ABB RobotStudio station: Assignment2_task#1.rsstn

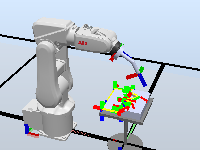
Station Assignment2_task#1 (saved by RobotStudio 20.1.9014.1)
Controller SystemTask1, task T_ROB1: task frame (RAPID world) sits at (150, 100, 0) mm in the station
Controller SystemTask1
  mechanical unit ROB_1: IRB120_3_58__01, 6 joints, base frame (0, 0, 0) mm
Layout (positions relative to the parent item):
  - IRB120_3_58__01 [mechanism, from Robots\IRB120_3_58_G_01.rslib] at (150, 100, 0) mm; joint values [0, 0, 0, 0, 0.5236, 0] (rad or m)
  - AssemblyWeldingTorch [part] at (452.8, 131.78, 541.25) mm, rotated rx -30 ry 0 rz -90 deg
  - Task1_Part1_2 [part] at (570, 0, 300) mm, rotated rx 90 ry 0 rz 0 deg
  - Task1_Part2 [part] at (470, 0, 300) mm, rotated rx 90 ry 0 rz 0 deg
  - Part_1 [part]
  - Part_2 [part]
  - Part_3 [part]
  - Part_4 [part]
Attachment: AssemblyWeldingTorch is attached to IRB120_3_58__01 / Link6
Attachment: Task1_Part2 is attached to Task1_Part1_2
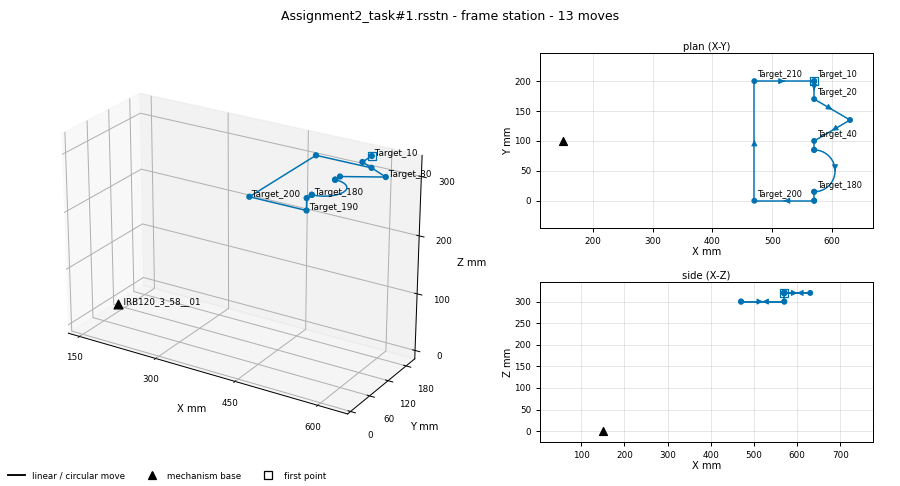
[picture p0: tool path of Assignment2_task#1.rsstn in frame station, 13 of 13 moves have a stored position in this frame; points joined in program order, loops and branches not executed]
Targets, tools, work objects and paths stored in the station, written as RAPID:
! task T_ROB1
MODULE CalibData
  TASK PERS tooldata WeldingTorch:=[TRUE,[[41,0,150.621],[0.965925826,0,0.258819045,0]],[1,[0,0,1],[1,0,0,0],0,0,0]];
  TASK PERS wobjdata Part1:=[FALSE,TRUE,"",[[420,-100,0],[0.707106781,0,0,0.707106781]],[[0,0,0],[1,0,0,0]]];
  TASK PERS wobjdata TableFrame:=[FALSE,TRUE,"",[[420,0,15],[0,0,1,0]],[[0,0,0],[1,0,0,0]]];
ENDMODULE

! task T_ROB1
MODULE Module1
  CONST robtarget Target_10:=[[0,100,-305],[0.707106781,0,0,-0.707106781],[0,0,0,0],[9E+09,9E+09,9E+09,9E+09,9E+09,9E+09]];
  CONST robtarget Target_20:=[[0,70,-305],[0.707106781,0,0,-0.707106781],[0,0,0,0],[9E+09,9E+09,9E+09,9E+09,9E+09,9E+09]];
  CONST robtarget Target_30:=[[-60,35,-305],[0.260979979,0,0,-0.965344213],[0,0,0,0],[9E+09,9E+09,9E+09,9E+09,9E+09,9E+09]];
  CONST robtarget Target_40:=[[0,0,-305],[0.965344213,0,0,-0.260979979],[0,0,0,0],[9E+09,9E+09,9E+09,9E+09,9E+09,9E+09]];
  CONST robtarget Target_50:=[[0,-15,-305],[0.707106781,0,0,-0.707106781],[0,0,0,0],[9E+09,9E+09,9E+09,9E+09,9E+09,9E+09]];
  CONST robtarget Target_60:=[[0,-15,-305],[0,0,0,1],[0,0,0,0],[9E+09,9E+09,9E+09,9E+09,9E+09,9E+09]];
  CONST robtarget Target_70:=[[-30.310889132,-32.5,-305],[0.5,0,0,-0.866025404],[0,0,0,0],[9E+09,9E+09,9E+09,9E+09,9E+09,9E+09]];
  CONST robtarget Target_80:=[[-30.310889132,-67.5,-305],[0.866025404,0,0,-0.5],[0,0,0,0],[9E+09,9E+09,9E+09,9E+09,9E+09,9E+09]];
  CONST robtarget Target_90:=[[0,-85,-305],[1,0,0,0],[0,0,0,0],[9E+09,9E+09,9E+09,9E+09,9E+09,9E+09]];
  CONST robtarget Target_100:=[[0,-85,-305],[0.707106781,0,0,-0.707106781],[0,0,0,0],[9E+09,9E+09,9E+09,9E+09,9E+09,9E+09]];
  CONST robtarget Target_110:=[[0,-100,-305],[0.707106781,0,0,-0.707106781],[0,0,0,0],[9E+09,9E+09,9E+09,9E+09,9E+09,9E+09]];
  CONST robtarget Target_120:=[[0,-100,-305],[0.5,-0.5,-0.5,-0.5],[0,0,0,0],[9E+09,9E+09,9E+09,9E+09,9E+09,9E+09]];
  CONST robtarget Target_130:=[[0,-100,-285],[0.5,-0.5,-0.5,-0.5],[0,0,0,0],[9E+09,9E+09,9E+09,9E+09,9E+09,9E+09]];
  CONST robtarget Target_140:=[[100,-100,-285],[1,0,0,0],[0,0,0,0],[9E+09,9E+09,9E+09,9E+09,9E+09,9E+09]];
  CONST robtarget Target_150:=[[100,100,-285],[0.707106781,0,0,0.707106781],[0,0,0,0],[9E+09,9E+09,9E+09,9E+09,9E+09,9E+09]];
  CONST robtarget Target_160:=[[0,-15,-305],[0,0,0,1],[0,0,0,0],[9E+09,9E+09,9E+09,9E+09,9E+09,9E+09]];
  CONST robtarget Target_170:=[[-35,-50,-305],[0.707106781,0,0,-0.707106781],[0,0,0,0],[9E+09,9E+09,9E+09,9E+09,9E+09,9E+09]];
  CONST robtarget Target_180:=[[0,-85,-305],[1,0,0,0],[0,0,0,0],[9E+09,9E+09,9E+09,9E+09,9E+09,9E+09]];
  CONST robtarget Target_190:=[[0,-100,-285],[0.707106781,-0.707106781,0,0],[0,0,0,0],[9E+09,9E+09,9E+09,9E+09,9E+09,9E+09]];
  CONST robtarget Target_200:=[[100,-100,-285],[0.707106781,-0.707106781,0,0],[0,0,0,0],[9E+09,9E+09,9E+09,9E+09,9E+09,9E+09]];
  CONST robtarget Target_210:=[[100,100,-285],[0.5,-0.5,-0.5,0.5],[0,0,0,0],[9E+09,9E+09,9E+09,9E+09,9E+09,9E+09]];
  CONST robtarget Target_220:=[[0,100,-285],[0,0,-0.707106781,0.707106781],[0,0,0,0],[9E+09,9E+09,9E+09,9E+09,9E+09,9E+09]];
  PROC main()
    Path_30;
  ENDPROC
  PROC Path_30()
    MoveL Target_10,v100,z10,WeldingTorch\WObj:=TableFrame;
    MoveL Target_20,v100,z10,WeldingTorch\WObj:=TableFrame;
    MoveL Target_30,v100,z10,WeldingTorch\WObj:=TableFrame;
    MoveL Target_40,v100,z10,WeldingTorch\WObj:=TableFrame;
    MoveL Target_50,v100,z10,WeldingTorch\WObj:=TableFrame;
    MoveL Target_160,v100,z10,WeldingTorch\WObj:=TableFrame;
    MoveC Target_170,Target_180,v100,z10,WeldingTorch\WObj:=TableFrame;
    MoveL Target_100,v100,z10,WeldingTorch\WObj:=TableFrame;
    MoveL Target_110,v100,z10,WeldingTorch\WObj:=TableFrame;
    MoveL Target_190,v100,z10,WeldingTorch\WObj:=TableFrame;
    MoveL Target_200,v100,z10,WeldingTorch\WObj:=TableFrame;
    MoveL Target_210,v100,z10,WeldingTorch\WObj:=TableFrame;
    MoveL Target_220,v100,z10,WeldingTorch\WObj:=TableFrame;
  ENDPROC
  PROC Path_40()
  ENDPROC
ENDMODULE

